ABB RAPID module: mdl.mod

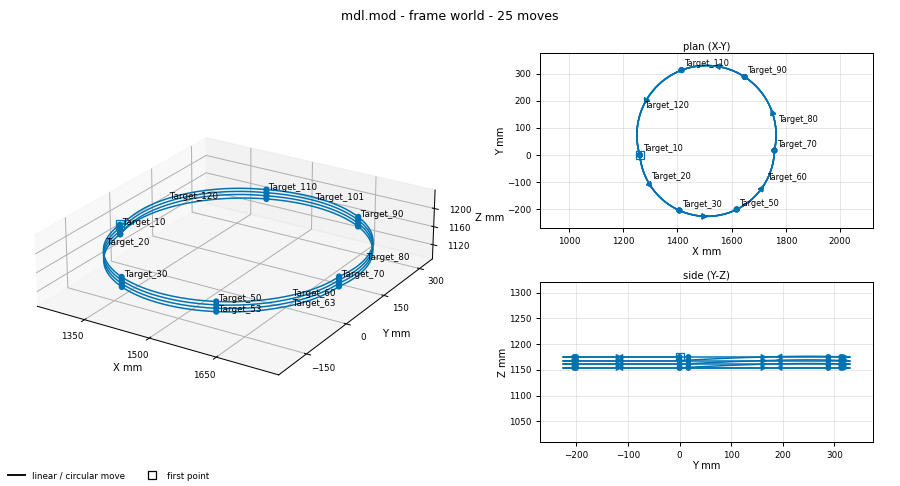
[picture p0: tool path of mdl.mod in frame world, 25 of 25 moves have a stored position in this frame; points joined in program order, loops and branches not executed]
MODULE Module1

    CONST robtarget Target_10:=[[1260.98395847,0,1175],[0.001103737,0,0.999999391,0],[0,0,0,0],[9E+09,9E+09,9E+09,9E+09,9E+09,9E+09]];
    CONST robtarget Target_20:=[[1292.592591169,-100.45010079,1175],[0.001100055,-0.000002723,0.999999395,0.000000346],[-1,0,-1,0],[9E+09,9E+09,9E+09,9E+09,9E+09,9E+09]];
    CONST robtarget Target_30:=[[1407.032853079,-204.29479274,1175],[0.001105033,0.000000768,0.999999389,-0.00000005],[-1,0,-1,0],[9E+09,9E+09,9E+09,9E+09,9E+09,9E+09]];
    CONST robtarget Target_40:=[[1539.046057366,-224.298691548,1175],[0.001103471,-0.000000018,0.999999391,-0.000000015],[-1,0,-1,0],[9E+09,9E+09,9E+09,9E+09,9E+09,9E+09]];
    CONST robtarget Target_50:=[[1618.6618035,-200.631421163,1175],[0.001103367,-0.000000045,0.999999391,0.000000214],[-1,0,-1,0],[9E+09,9E+09,9E+09,9E+09,9E+09,9E+09]];
    CONST robtarget Target_60:=[[1721.924358011,-106.035265256,1175],[0.00110325,-0.000000461,0.999999391,0.000000173],[-1,0,-1,0],[9E+09,9E+09,9E+09,9E+09,9E+09,9E+09]];
    CONST robtarget Target_70:=[[1757.807980431,17.128948752,1175],[0.001103223,-0.000000018,0.999999391,-0.000000016],[0,-1,0,0],[9E+09,9E+09,9E+09,9E+09,9E+09,9E+09]];
    CONST robtarget Target_80:=[[1761.633768624,108.810266112,1175],[0.001101579,0.000000003,0.999999393,-0.000000109],[0,-1,0,0],[9E+09,9E+09,9E+09,9E+09,9E+09,9E+09]];
    CONST robtarget Target_90:=[[1648.139955341,288.428493111,1175],[0.001104242,0.000004916,0.99999939,-0.000001118],[0,-1,0,0],[9E+09,9E+09,9E+09,9E+09,9E+09,9E+09]];
    CONST robtarget Target_100:=[[1517.367949203,330.304204057,1175],[0.001103041,-0.000000017,0.999999392,-0.000000023],[0,-1,0,0],[9E+09,9E+09,9E+09,9E+09,9E+09,9E+09]];
    CONST robtarget Target_110:=[[1414.931656149,313.355759543,1175],[0.001104985,-0.00000091,0.99999939,-0.000000046],[0,-1,0,0],[9E+09,9E+09,9E+09,9E+09,9E+09,9E+09]];
    CONST robtarget Target_120:=[[1265.773979419,161.604103504,1175],[0.001103546,0.000000104,0.999999391,-0.000000179],[0,-1,0,0],[9E+09,9E+09,9E+09,9E+09,9E+09,9E+09]];



    CONST robtarget Target_11:=[[1260.98395847,0,1168],[0.001103737,0,0.999999391,0],[0,0,0,0],[9E+09,9E+09,9E+09,9E+09,9E+09,9E+09]];
    CONST robtarget Target_21:=[[1292.592591169,-100.45010079,1168],[0.001100055,-0.000002723,0.999999395,0.000000346],[-1,0,-1,0],[9E+09,9E+09,9E+09,9E+09,9E+09,9E+09]];
    CONST robtarget Target_31:=[[1407.032853079,-204.29479274,1168],[0.001105033,0.000000768,0.999999389,-0.00000005],[-1,0,-1,0],[9E+09,9E+09,9E+09,9E+09,9E+09,9E+09]];
    CONST robtarget Target_41:=[[1539.046057366,-224.298691548,1168],[0.001103471,-0.000000018,0.999999391,-0.000000015],[-1,0,-1,0],[9E+09,9E+09,9E+09,9E+09,9E+09,9E+09]];
    CONST robtarget Target_51:=[[1618.6618035,-200.631421163,1168],[0.001103367,-0.000000045,0.999999391,0.000000214],[-1,0,-1,0],[9E+09,9E+09,9E+09,9E+09,9E+09,9E+09]];
    CONST robtarget Target_61:=[[1721.924358011,-106.035265256,1168],[0.00110325,-0.000000461,0.999999391,0.000000173],[-1,0,-1,0],[9E+09,9E+09,9E+09,9E+09,9E+09,9E+09]];
    CONST robtarget Target_71:=[[1757.807980431,17.128948752,1168],[0.001103223,-0.000000018,0.999999391,-0.000000016],[0,-1,0,0],[9E+09,9E+09,9E+09,9E+09,9E+09,9E+09]];
    CONST robtarget Target_81:=[[1761.633768624,108.810266112,1168],[0.001101579,0.000000003,0.999999393,-0.000000109],[0,-1,0,0],[9E+09,9E+09,9E+09,9E+09,9E+09,9E+09]];
    CONST robtarget Target_91:=[[1648.139955341,288.428493111,1168],[0.001104242,0.000004916,0.99999939,-0.000001118],[0,-1,0,0],[9E+09,9E+09,9E+09,9E+09,9E+09,9E+09]];
    CONST robtarget Target_101:=[[1517.367949203,330.304204057,1168],[0.001103041,-0.000000017,0.999999392,-0.000000023],[0,-1,0,0],[9E+09,9E+09,9E+09,9E+09,9E+09,9E+09]];
    CONST robtarget Target_111:=[[1414.931656149,313.355759543,1168],[0.001104985,-0.00000091,0.99999939,-0.000000046],[0,-1,0,0],[9E+09,9E+09,9E+09,9E+09,9E+09,9E+09]];
    CONST robtarget Target_121:=[[1265.773979419,161.604103504,1168],[0.001103546,0.000000104,0.999999391,-0.000000179],[0,-1,0,0],[9E+09,9E+09,9E+09,9E+09,9E+09,9E+09]];

    CONST robtarget Target_12:=[[1260.98395847,0,1161],[0.001103737,0,0.999999391,0],[0,0,0,0],[9E+09,9E+09,9E+09,9E+09,9E+09,9E+09]];
    CONST robtarget Target_22:=[[1292.592591169,-100.45010079,1161],[0.001100055,-0.000002723,0.999999395,0.000000346],[-1,0,-1,0],[9E+09,9E+09,9E+09,9E+09,9E+09,9E+09]];
    CONST robtarget Target_32:=[[1407.032853079,-204.29479274,1161],[0.001105033,0.000000768,0.999999389,-0.00000005],[-1,0,-1,0],[9E+09,9E+09,9E+09,9E+09,9E+09,9E+09]];
    CONST robtarget Target_42:=[[1539.046057366,-224.298691548,1161],[0.001103471,-0.000000018,0.999999391,-0.000000015],[-1,0,-1,0],[9E+09,9E+09,9E+09,9E+09,9E+09,9E+09]];
    CONST robtarget Target_52:=[[1618.6618035,-200.631421163,1161],[0.001103367,-0.000000045,0.999999391,0.000000214],[-1,0,-1,0],[9E+09,9E+09,9E+09,9E+09,9E+09,9E+09]];
    CONST robtarget Target_62:=[[1721.924358011,-106.035265256,1161],[0.00110325,-0.000000461,0.999999391,0.000000173],[-1,0,-1,0],[9E+09,9E+09,9E+09,9E+09,9E+09,9E+09]];
    CONST robtarget Target_72:=[[1757.807980431,17.128948752,1161],[0.001103223,-0.000000018,0.999999391,-0.000000016],[0,-1,0,0],[9E+09,9E+09,9E+09,9E+09,9E+09,9E+09]];
    CONST robtarget Target_82:=[[1761.633768624,108.810266112,1161],[0.001101579,0.000000003,0.999999393,-0.000000109],[0,-1,0,0],[9E+09,9E+09,9E+09,9E+09,9E+09,9E+09]];
    CONST robtarget Target_92:=[[1648.139955341,288.428493111,1161],[0.001104242,0.000004916,0.99999939,-0.000001118],[0,-1,0,0],[9E+09,9E+09,9E+09,9E+09,9E+09,9E+09]];
    CONST robtarget Target_102:=[[1517.367949203,330.304204057,1161],[0.001103041,-0.000000017,0.999999392,-0.000000023],[0,-1,0,0],[9E+09,9E+09,9E+09,9E+09,9E+09,9E+09]];
    CONST robtarget Target_112:=[[1414.931656149,313.355759543,1161],[0.001104985,-0.00000091,0.99999939,-0.000000046],[0,-1,0,0],[9E+09,9E+09,9E+09,9E+09,9E+09,9E+09]];
    CONST robtarget Target_122:=[[1265.773979419,161.604103504,1161],[0.001103546,0.000000104,0.999999391,-0.000000179],[0,-1,0,0],[9E+09,9E+09,9E+09,9E+09,9E+09,9E+09]];

    CONST robtarget Target_13:=[[1260.98395847,0,1154],[0.001103737,0,0.999999391,0],[0,0,0,0],[9E+09,9E+09,9E+09,9E+09,9E+09,9E+09]];
    CONST robtarget Target_23:=[[1292.592591169,-100.45010079,1154],[0.001100055,-0.000002723,0.999999395,0.000000346],[-1,0,-1,0],[9E+09,9E+09,9E+09,9E+09,9E+09,9E+09]];
    CONST robtarget Target_33:=[[1407.032853079,-204.29479274,1154],[0.001105033,0.000000768,0.999999389,-0.00000005],[-1,0,-1,0],[9E+09,9E+09,9E+09,9E+09,9E+09,9E+09]];
    CONST robtarget Target_43:=[[1539.046057366,-224.298691548,1154],[0.001103471,-0.000000018,0.999999391,-0.000000015],[-1,0,-1,0],[9E+09,9E+09,9E+09,9E+09,9E+09,9E+09]];
    CONST robtarget Target_53:=[[1618.6618035,-200.631421163,1154],[0.001103367,-0.000000045,0.999999391,0.000000214],[-1,0,-1,0],[9E+09,9E+09,9E+09,9E+09,9E+09,9E+09]];
    CONST robtarget Target_63:=[[1721.924358011,-106.035265256,1154],[0.00110325,-0.000000461,0.999999391,0.000000173],[-1,0,-1,0],[9E+09,9E+09,9E+09,9E+09,9E+09,9E+09]];
    CONST robtarget Target_73:=[[1757.807980431,17.128948752,1154],[0.001103223,-0.000000018,0.999999391,-0.000000016],[0,-1,0,0],[9E+09,9E+09,9E+09,9E+09,9E+09,9E+09]];
    CONST robtarget Target_83:=[[1761.633768624,108.810266112,1154],[0.001101579,0.000000003,0.999999393,-0.000000109],[0,-1,0,0],[9E+09,9E+09,9E+09,9E+09,9E+09,9E+09]];
    CONST robtarget Target_93:=[[1648.139955341,288.428493111,1154],[0.001104242,0.000004916,0.99999939,-0.000001118],[0,-1,0,0],[9E+09,9E+09,9E+09,9E+09,9E+09,9E+09]];
    CONST robtarget Target_103:=[[1517.367949203,330.304204057,1154],[0.001103041,-0.000000017,0.999999392,-0.000000023],[0,-1,0,0],[9E+09,9E+09,9E+09,9E+09,9E+09,9E+09]];
    CONST robtarget Target_113:=[[1414.931656149,313.355759543,1154],[0.001104985,-0.00000091,0.99999939,-0.000000046],[0,-1,0,0],[9E+09,9E+09,9E+09,9E+09,9E+09,9E+09]];
    CONST robtarget Target_123:=[[1265.773979419,161.604103504,1154],[0.001103546,0.000000104,0.999999391,-0.000000179],[0,-1,0,0],[9E+09,9E+09,9E+09,9E+09,9E+09,9E+09]];

    !***********************************************************
    !
    ! Module:  Module1
    !
    ! Description:
    !   <Insert description here>
    !
    ! Author: cvv2278
    !
    ! Version: 1.0
    !
    !***********************************************************


    !***********************************************************
    !
    ! Procedure main
    !
    !   This is the entry point of your program
    !
    !***********************************************************
    PROC main()
        Path_10;
    ENDPROC

    PROC Path_10()
        MoveJ Target_10,v1000,fine,MyTool\WObj:=wobj0;
        MoveC Target_20,Target_30,v1000,z20,MyTool\WObj:=wobj0;
        MoveC Target_40,Target_50,v1000,z20,MyTool\WObj:=wobj0;
        MoveC Target_60,Target_70,v1000,z20,MyTool\WObj:=wobj0;
        MoveC Target_80,Target_90,v1000,z20,MyTool\WObj:=wobj0;
        MoveC Target_100,Target_110,v1000,z20,MyTool\WObj:=wobj0;

        MoveC Target_120, Target_11,v1000,z20,MyTool\WObj:=wobj0;
        MoveC Target_21,Target_31,v1000,z20,MyTool\WObj:=wobj0;
        MoveC Target_41,Target_51,v1000,z20,MyTool\WObj:=wobj0;
        MoveC Target_61,Target_71,v1000,z20,MyTool\WObj:=wobj0;
        MoveC Target_81,Target_91,v1000,z20,MyTool\WObj:=wobj0;
        MoveC Target_101,Target_111,v1000,z20,MyTool\WObj:=wobj0;


        MoveC Target_121, Target_12,v1000,z20,MyTool\WObj:=wobj0;
        MoveC Target_22,Target_32,v1000,z20,MyTool\WObj:=wobj0;
        MoveC Target_42,Target_52,v1000,z20,MyTool\WObj:=wobj0;
        MoveC Target_62,Target_72,v1000,z20,MyTool\WObj:=wobj0;
        MoveC Target_82,Target_92,v1000,z20,MyTool\WObj:=wobj0;
        MoveC Target_102,Target_112,v1000,z20,MyTool\WObj:=wobj0;


        MoveC Target_122, Target_13,v1000,z20,MyTool\WObj:=wobj0;
        MoveC Target_23,Target_33,v1000,z20,MyTool\WObj:=wobj0;
        MoveC Target_43,Target_53,v1000,z20,MyTool\WObj:=wobj0;
        MoveC Target_63,Target_73,v1000,z20,MyTool\WObj:=wobj0;
        MoveC Target_83,Target_93,v1000,z20,MyTool\WObj:=wobj0;
        MoveC Target_103,Target_113,v1000,z20,MyTool\WObj:=wobj0;
        MoveC Target_123,Target_13,v1000,fine,MyTool\WObj:=wobj0;

    ENDPROC
ENDMODULE
